// TIA Portal V19 export
TYPE "LAF_typeSequenceCommands"
TITLE = typeEquipmentA_Interface
// Commands for the sequence
// stored: Access Published
   STRUCT
      setAutomaticMode : Bool;   // Set to Automatic Mode
      setSingleStepMode : Bool;   // Set to Single Step Mode
      off : Bool;   // Turn sequence off, deactivate all steps
      initialize : Bool;   // Go to IDLE step
      start : Bool;   // Start condition to gro from IDLE to first process step
      immediateStop : Bool;   // Go to IMMEDIATE_STOP step
      hold : Bool;   // Pause state machine after current step completed
      nextStep : Bool;   // Go to next step (if SingleStep mode is active)
      interlockStepChange : Bool;   // Prevent going to next step
   END_STRUCT;
END_TYPE
